(* IEC 61131-3 sources: repo_PLC_code_eval/dataset/2021-8-20/F05_系统操作, 1 file *)

(* ---- Fun_系统停止.st ---- *)
FUNCTION Fun_系统停止 : DWORD
VAR_IN_OUT
	EventPrm: CmpApp.EVTPARAM_CmpAppStop;
END_VAR
VAR
END_VAR
